PROGRAM P17_DOROperation
VAR_INPUT
	bDOROn				: BOOL; //UI Input Button
	bDOROff				: BOOL; //UI Input Button
	fTresholdPressure	: REAL;
	fTresholdCount		: REAL;
	bPressureEnable 	: BOOL;
	bCountEnable		: BOOL;
END_VAR
VAR_OUTPUT
	isDOROnState		: BOOL := FALSE; //DOR ON State
	bError				: INT; //0: No Err, 1: Vacuum Fail, 2: Vacuum Release, 3: Try out
	nWaitCounter		: INT;
END_VAR
VAR
	(* Input *)
	bVacSwitch			: BOOL; //Push Switch
	bAtmSwitch			: BOOL; //Push Switch
	(* Pressure Transducer *)
	nPressurePV			: INT;
	rPressurePV_kPa		: REAL;
	(* Output *)
	bVacLED				: BOOL;
	bAtmLED				: BOOL;
	bV_DORVac			: BOOL; //V34 Valve
	bV_DORFill			: BOOL; //V35 Valve
	
	(* DOR Condition Operation Parameter *)
	rTrigSwitch			: R_TRIG;
	TimerOnLED			: TON;
	TimerVacSwitch		: TON;
	TimerAtmSwitch		: TON;
	TimerWaitCheck		: TON;
	TimerVacRealease	: TON;
	nCase				: INT := 0;
	nTresholdCount		: INT;
	nTryCount			: INT;
	bVacuumRealse		: BOOL;
	//Temperatur Variable
	bTest				: BOOL;
	nTest				: INT;
END_VAR

VAR CONSTANT
	KL3464MaxValueP		: REAL := 16383; //1 ~ 5VDC, 0 ~ 100kPa(1bar), PG35
	SlopeFactor			: REAL := 0.007617887; //100kPa/(16383-3256)
END_VAR

// Double O-Ring Vacuum Condition

(* Read from Device Value *)
// DOR Operation Switch
bVacSwitch 			:= GVL_IO.aDigitalInputIO[1].4; //Switch Input
bAtmSwitch 			:= GVL_IO.aDigitalInputIO[1].5; //Switch Input
nPressurePV 		:= GVL_IO.aAnalogInputIO[29];
rPressurePV_kPa 	:= (nPressurePV-3256)*SlopeFactor;

fTresholdPressure 	:= GVL_IO.aInterlockSet[15];
fTresholdCount 		:= GVL_IO.aInterlockSet[16];
bPressureEnable 	:= GVL_IO.aInterlockEnable[1].5;
bCountEnable 		:= GVL_IO.aInterlockEnable[1].6;
nTresholdCount 		:= REAL_TO_INT(fTresholdCount); //Try One more Vacuum 
(* If Vacuum 'ON' Switch Press, Change DOR Vacuum State *)
//DOR Operation Signal generation
TimerVacSwitch(IN:=bVacSwitch OR bDOROn, PT:=T#100MS);
rTrigSwitch(CLK:=TimerVacSwitch.Q);

IF rTrigSwitch.Q AND P90_Interlock.bDorOnEnable THEN
	nCase 		:= 1;
	nTryCount 	:= 1; //Try One more Vacuum 
END_IF

CASE nCase OF
	1: //Initialize
		isDOROnState := FALSE;
		bV_DORVac 	:= TRUE; //V34 Open
		bV_DORFill	:= FALSE; //V35 Close
		bAtmLED		:= FALSE;
		TimerWaitCheck(IN:=FALSE);	
		nCase := 10;
	10: //Wait and Vacuum Check
		(* Blink Switch LED *)
		TimerOnLED(IN:=TRUE, PT:=T#500MS);
		IF TimerOnLED.Q THEN
			TimerOnLED(IN:=FALSE);
			bVacLED := NOT(bVacLED);
		END_IF

		TimerWaitCheck(IN:=TRUE, PT:=T#5S);
		IF TimerWaitCheck.Q THEN
			IF rPressurePV_kPa > fTresholdPressure THEN
				bV_DORVac 		:= FALSE; //V34 Close
				isDOROnState 	:= TRUE;
				bVacLED 			:= TRUE; //Switch LED
				bError			:= 0;
				nCase 			:= 0;
			ELSIF nTryCount < nTresholdCount THEN
				TimerWaitCheck(IN:=FALSE);
				nTryCount 		:= nTryCount + 1;				
				nCase 			:= 1;
			ELSE
				bV_DORVac 		:= FALSE; //V34 Close
				isDOROnState 	:= FALSE;
				bVacLED			:= FALSE; //Switch LED
				bError			:= 1; // Vacuum Fail
				nCase			:= 0;
			END_IF
		END_IF
END_CASE

(* If Vacuum 'OFF' Switch Press, Change DOR Vent(Fill, Atm) State *)
//DOR Operation Signal generation
TimerAtmSwitch(IN:=bAtmSwitch OR bDOROff, PT:=T#100MS);
rTrigSwitch(CLK:=TimerAtmSwitch.Q);

IF rTrigSwitch.Q AND P90_Interlock.bDorOffEnable THEN
	nCase := 2;
END_IF

CASE nCase OF
	2:
		(* Blink Switch LED *)
		TimerOnLED(IN:=TRUE, PT:=T#500MS);
		IF TimerOnLED.Q THEN
			TimerOnLED(IN:=FALSE);
			bAtmLED := NOT(bAtmLED);
		END_IF
		
		TimerWaitCheck(IN:=TRUE, PT:=T#10S);
		nWaitCounter := TIME_TO_INT(TimerWaitCheck.ET/1000);
		IF TimerWaitCheck.Q THEN
			TimerWaitCheck(IN:=FALSE);
			bVacLED			:= FALSE;
			bV_DORVac 		:= FALSE; //V34 Close
			bV_DORFill		:= TRUE; //V35 Open
			nCase			:= 20;
		END_IF
	20:
		TimerWaitCheck(IN:=TRUE, PT:=T#5S);
		IF TimerWaitCheck.Q THEN
			bVacLED			:= FALSE;
			bV_DORFill		:= FALSE;
			isDOROnState 	:= FALSE;
			bAtmLED			:= TRUE;
			nCase			:= 0;
		END_IF
END_CASE

(* If Vacuum 'ON' State, Check the Vacuum range *)
IF isDOROnState AND rPressurePV_kPa < (fTresholdPressure - 20) AND nTryCount < 3 THEN
	bError := 2; // Vacuum release
	TimerVacRealease(IN:=TRUE, PT:=T#2S);
	
	(* Blink Vac Switch LED *)
	TimerOnLED(IN:=TRUE, PT:=T#500MS);
	IF TimerOnLED.Q THEN
		TimerOnLED(IN:=FALSE);
		bVacLED := NOT(bVacLED);
	END_IF

	IF TimerVacRealease.Q  THEN
		TimerVacRealease(IN:=FALSE);
		nTryCount 		:= nTryCount + 1;
		bV_DORVac 		:= FALSE;//Vacuum Valve OFF
		bVacLED := TRUE;
	ELSE
		bV_DORVac 		:= TRUE;//Vacuum Valve ON
	END_IF
	
ELSIF bError = 2 THEN
	bV_DORVac := FALSE;
	bError := 0;
	
ELSIF nTryCount >= 3 THEN
	bV_DORVac := FALSE;
	bError := 3; //Vacuum Released
END_IF

//알람 리셋
IF GVL_IO.aInterlockEnable[1].0 OR GVL_IO.aInterlockEnable[1].1 THEN
	bError := 0;
END_IF

(* Write to Device Value *)
// Cover Operation Switch Lamp
GVL_IO.aOutputSolValve[2].18 := bV_DORVac; //V34
GVL_IO.aOutputSolValve[2].19 := bV_DORFill; //V35
GVL_IO.aDigitalOutputIO[4].0 := bVacLED;
GVL_IO.aDigitalOutputIO[4].1 := bAtmLED;

END_PROGRAM

(* stored: Version 1.1.0.1, ProductVersion 3.1.4026.11
   POU P17_DOROperation: Id {47a43ac8-2dfa-477f-bf65-90da71792e7e}, SpecialFunc None *)
